{attribute 'c++_compatible'}
FUNCTION_BLOCK FB_UdpClientRT IMPLEMENTS ITcIoUdpProtocolRecv
VAR_INPUT
	
END_VAR
VAR_OUTPUT
END_VAR
VAR
	// ITcIoUdpProtocolRecv related 
	{attribute 'TcInitSymbol'}
	oid : OTCID; 
	ipUdp : ITcIoUdpProtocol;
	
	// Initilized variables
	remoteIpAddr : UDINT;
	remotePort : UINT;
	localPort : UINT;
	{attribute 'tc_no_symbol'}
	nRxData : UDINT := 0;
	{attribute 'tc_no_symbol'}
	pRxData : PVOID;
	{attribute 'tc_no_symbol'}
	nTxData : UDINT := 0;
	{attribute 'tc_no_symbol'}
	pTxData : PVOID;
	
	// Send/Recv counters
	rxCounter : UINT;
	txCounter : UINT;
	
	// Result
	hrInit : HRESULT;
	hrSend : HRESULT;
END_VAR

IF ipUdp <> 0 THEN
	// Send data to remote server
	IF nTxData > 0 THEN		
		hrSend := ipUdp.SendData(remoteIpAddr, remotePort, localPort, nTxData, pTxData, TRUE, 0);
		txCounter := txCounter + 1;
	END_IF
	
	// Check for incoming data
	IF nRxData > 0 THEN
		ipUdp.CheckReceived();
	END_IF
END_IF

{attribute 'conditionalshow'}
METHOD FB_exit : BOOL
VAR_INPUT
	bInCopyCode : BOOL; // if TRUE, the exit method is called for exiting an instance that is copied afterwards (online change).
END_VAR
IF NOT bInCopyCode THEN // no online change
	IF ipUdp <> 0 THEN 
		ipUdp.UnregisterReceiver(localPort); // Shutdown
		FW_SafeRelease(ADR(ipUdp));
		FB_exit := TRUE; 
	END_IF
END_IF
END_METHOD

{attribute 'conditionalshow'}
METHOD FB_init : BOOL
VAR_INPUT
	bInitRetains : BOOL; // if TRUE, the retain variables are initialized (warm start / cold start)
	bInCopyCode : BOOL;  // if TRUE, the instance afterwards gets moved into the copy code (online change)
	
	// Init variables
	_remoteIpAddr : T_Ipv4Addr;
	_remotePort : UINT;
	_localPort : UINT;
	_nRxData : UDINT;
	_pRxData : PVOID;
	_nTxData : UDINT;
	_pTxData : PVOID;
END_VAR
VAR
    ipSrv : ITComObjectServer;
	ipArr : T_IPv4AddrArr;
	i : UINT;
END_VAR
// Initilize member variables
remoteIpAddr := IpToLong(_remoteIpAddr);
remotePort := _remotePort;
localPort := _localPort;
nRxData := _nRxData;
pRxData := _pRxData;
nTxData := _nTxData;
pTxData := _pTxData;

IF NOT bInCopyCode THEN // no online change
	IF ipUdp = 0 THEN
	    hrInit := FW_ObjMgr_GetObjectInstance(
			oid:=oid, 
			iid:=TC_GLOBAL_IID_LIST.IID_ITcIoUdpProtocol, 
			pipUnk:=ADR(ipUdp)
		);
		
		IF SUCCEEDED(hrInit) THEN 
			IF  SUCCEEDED(ipUdp.RegisterReceiver(localPort, THIS^)) THEN //open port
				FB_init := TRUE;
			ELSE 
				FW_SafeRelease(ADR(ipUdp));
			END_IF
		END_IF				
	END_IF
END_IF
END_METHOD

{attribute 'conditionalshow'}
METHOD FB_reinit : BOOL
VAR_INPUT
END_VAR
IF (ipUdp <> 0) THEN 
	ipUdp.RegisterReceiver(localPort, THIS^);
	FB_reinit := TRUE; 
END_IF
END_METHOD

METHOD IpToLong : UDINT
VAR_INPUT
	ipAddr : T_Ipv4Addr;
END_VAR

VAR
	ipAddrArr : T_Ipv4AddrArr;
	ipAddrLong : UDINT;
END_VAR
// Scan ip string to byte array
ipAddrArr := F_ScanIPv4AddrIds(ipAddr);

// Copy bytes to ipaddrLong in reverse direction
MEMCPY(ADR(ipAddrLong) + 0, ADR(ipAddrArr) + 3, 1);
MEMCPY(ADR(ipAddrLong) + 1, ADR(ipAddrArr) + 2, 1);
MEMCPY(ADR(ipAddrLong) + 2, ADR(ipAddrArr) + 1, 1);
MEMCPY(ADR(ipAddrLong) + 3, ADR(ipAddrArr) + 0, 1); 

// Return long ip adress
IpToLong := ipAddrLong;
END_METHOD

{attribute 'object_name' := 'ReceiveData'}
{attribute 'c++_compatible'}
{attribute 'signature_flag' := '33554688'}
{attribute 'pack_mode' := '4'}
{attribute 'show'}
{attribute 'minimal_input_size' := '4'}
METHOD ReceiveData : HRESULT
VAR_INPUT
	ipAddr	: UDINT;
	udpDestPort	: UINT;
	udpSrcPort	: UINT;
	nData	: UDINT;
	pData	: PVOID;
	pVlan	: POINTER TO ETYPE_VLAN_HEADER := 0;
END_VAR
// Check data size and copy data
IF nData = nRxData THEN
	// Copy recived data
	MEMCPY(pRxData, pData, nRxData);
	
	// Increment counters
	rxCounter := rxCounter + 1;
END_IF
END_METHOD

{attribute 'object_name' := 'TcAddRef'}
{attribute 'c++_compatible'}
{attribute 'signature_flag' := '33554688'}
{attribute 'pack_mode' := '4'}
{attribute 'show'}
{attribute 'minimal_input_size' := '4'}
METHOD TcAddRef : UDINT
END_METHOD

{attribute 'object_name' := 'TcQueryInterface'}
{attribute 'c++_compatible'}
{attribute 'signature_flag' := '33554688'}
{attribute 'pack_mode' := '4'}
{attribute 'show'}
{attribute 'minimal_input_size' := '4'}
METHOD TcQueryInterface : HRESULT
VAR_INPUT
	iid	: REFERENCE TO IID;
	pipItf	: POINTER TO PVOID;
END_VAR
VAR
	ipUdpRecv : ITcIoUdpProtocolRecv;
	ipUnknown : ITcUnknown;	
END_VAR
IF GuidsEqual(ADR(iid), ADR(TC_GLOBAL_IID_LIST.IID_ITcIoUdpProtocolRecv)) THEN
	ipUdpRecv := THIS^; // cast to interface pointer
	pipItf^ := ITCUNKNOWN_TO_PVOID(ipUdpRecv);
	TcAddRef();
	TcQueryInterface := S_OK;
ELSIF GuidsEqual(ADR(iid), ADR(TC_GLOBAL_IID_LIST.IID_ITcUnknown)) THEN
	ipUnknown := THIS^; // cast to interface pointer
	pipItf^ := ITCUNKNOWN_TO_PVOID(ipUnknown);
	TcAddRef();
	TcQueryInterface := S_OK;
ELSE
	TcQueryInterface := E_HRESULTAdsErr.NOINTERFACE ; //Call super if this fb extends some other
END_IF
END_METHOD

{attribute 'object_name' := 'TcRelease'}
{attribute 'c++_compatible'}
{attribute 'signature_flag' := '33554688'}
{attribute 'pack_mode' := '4'}
{attribute 'show'}
{attribute 'minimal_input_size' := '4'}
METHOD TcRelease : UDINT
END_METHOD

END_FUNCTION_BLOCK

(* stored: Version 1.1.0.1, ProductVersion 3.1.4022.18
   POU FB_UdpClientRT: Id {a471e0e0-6cc0-46b7-a06a-91d73ef548ff}, SpecialFunc None
   Method FB_exit: Id {ce81e3ec-e82a-48c2-88e4-63c9532c782c}
   Method FB_init: Id {416426b6-cdda-48f2-b64a-9b8fd8f46e82}
   Method FB_reinit: Id {99272707-3866-4d48-957e-3b19210a87e8}
   Method IpToLong: Id {e4cca66b-0819-484f-a8e6-83fc33d50f23}
   Method ReceiveData: Id {e94ea7b4-e895-4e8d-84f8-a532daf3880f}
   Method TcAddRef: Id {e1334eda-f68a-4004-ab3f-36fe7d61d154}
   Method TcQueryInterface: Id {aab6f97f-6c35-4d15-aaf4-d9c9e8dffc1e}
   Method TcRelease: Id {c290f852-e38c-4827-82d1-07132089bfd0} *)
